TYPE DUT_HMI_14_MANUALS :
STRUCT
	PS : ARRAY[0..CNC.NUM_MAX_MANUALS_14-1] OF BOOL;
	LS : ARRAY[0..CNC.NUM_MAX_MANUALS_14-1] OF BOOL;
END_STRUCT
END_TYPE

(* stored: Version 1.1.0.1, ProductVersion 3.1.4024.13
   DUT DUT_HMI_14_MANUALS: Id {5d16d6e1-ff6c-4d6d-839e-8e001e930aaa} *)
